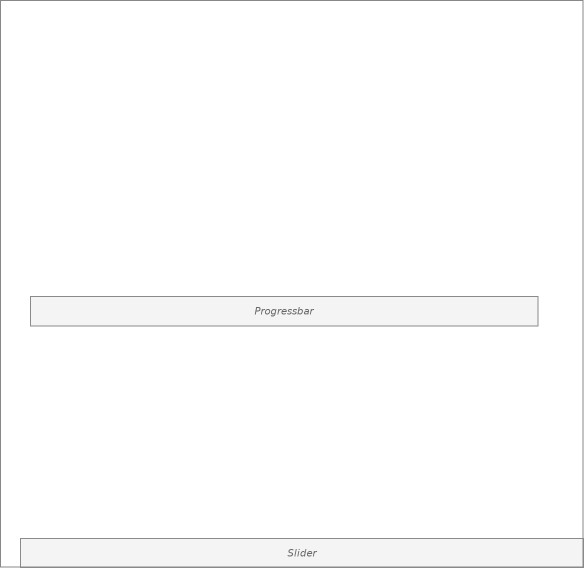
VISUALIZATION Visu  // 584x568
    Slider (20,538 564x30), variable: MAIN.nPmeter, scale 0..32767
    Progressbar (30,296 508x30), variable: MAIN.nValue
END_VISUALIZATION

(* stored: Version 1.1.0.1, ProductVersion 3.1.4024.12
   Visu Visu: Id {d603df1b-35b1-4fbd-9a8a-f3b8b10d3a23} *)
